(*

.. <legal notes>

legal notes
=================
| SPDX-FileCopyrightText: © 2026 Oleksandr Tiutyk <trofimich@gmail.com>
| SPDX-License-Identifier: LGPL-3.0-only
| For details check: LGPL-3.0-only_

.. _LGPL-3.0-only: https://www.gnu.org/licenses/lgpl-3.0.en.html

.. </legal notes>

*)

PROGRAM Trigonometry
VAR
	_ClassName : STRING := __POUNAME();

	_Random : DRAND;
END_VAR

{attribute 'monitoring' := 'call'}
PROPERTY ClassName : STRING
GET
ClassName := _ClassName;
END_GET
END_PROPERTY

METHOD ConvertDegreesToRadians : LREAL
VAR_INPUT
	degrees : LREAL;
END_VAR
ConvertDegreesToRadians := degrees * Tc2_System.Global_Variables.PI / 180;
END_METHOD

METHOD ConvertRadiansToDegrees : LREAL
VAR_INPUT
	radians : LREAL;
END_VAR
ConvertRadiansToDegrees := radians * 180 / Tc2_System.Global_Variables.PI;
END_METHOD

{attribute 'monitoring' := 'call'}
PROPERTY NamespaceName : STRING
GET
NamespaceName := CurrentNamespace.Name;
END_GET
END_PROPERTY

END_PROGRAM

(* stored: Version 1.1.0.1
   POU Trigonometry: Id {ae570430-0788-4098-b5e9-35c83e020aed}, SpecialFunc None
   Property ClassName: Id {264f7bce-b5ad-4665-b3b2-c4de52b54881}
   Get Get: Id {1e395fac-98c9-4834-8f6c-3003828075d8}
   Method ConvertDegreesToRadians: Id {af1fdb21-c3e3-4758-8c86-196812b69db4}
   Method ConvertRadiansToDegrees: Id {d7982d69-d3f1-4563-b861-3b474bd831ee}
   Property NamespaceName: Id {36f9cbaf-53f1-43d5-b546-e16c5138b6f4}
   Get Get: Id {c6133c90-814d-4fa4-ba08-b55048ab9e25} *)
